PROGRAM MAIN
VAR
	// Control Buttons
	ManualSwitch: BOOL;
	AutoSwitch: BOOL;
	AutoStartButton: BOOL;
	ForwardSwitch: BOOL;
	ReverseSwitch: BOOL;
	StopSwitch: BOOL;
	
	// Limit switches
	LimitSwitchRight: BOOL;
	LimitSwitchLeft: BOOL;
	
	// Operation modes
	ManualMode: BOOL;
	AutoMode: BOOL;
	AutoStart: BOOL;
	ManualForward: BOOL;
	ManualReverse: BOOL;
	ConfirmAutoForward: BOOL;
	AutoForward: BOOL;
	AutoReverse: BOOL;
	
	// Output coils
	MotorForward: BOOL;
	MotorReverse: BOOL;
	
	// Aux. blocks
	tonForward: TON;
END_VAR
VAR // added by the converter: edge detectors and wires of the graphical bodies
    _w1 : BOOL;
END_VAR

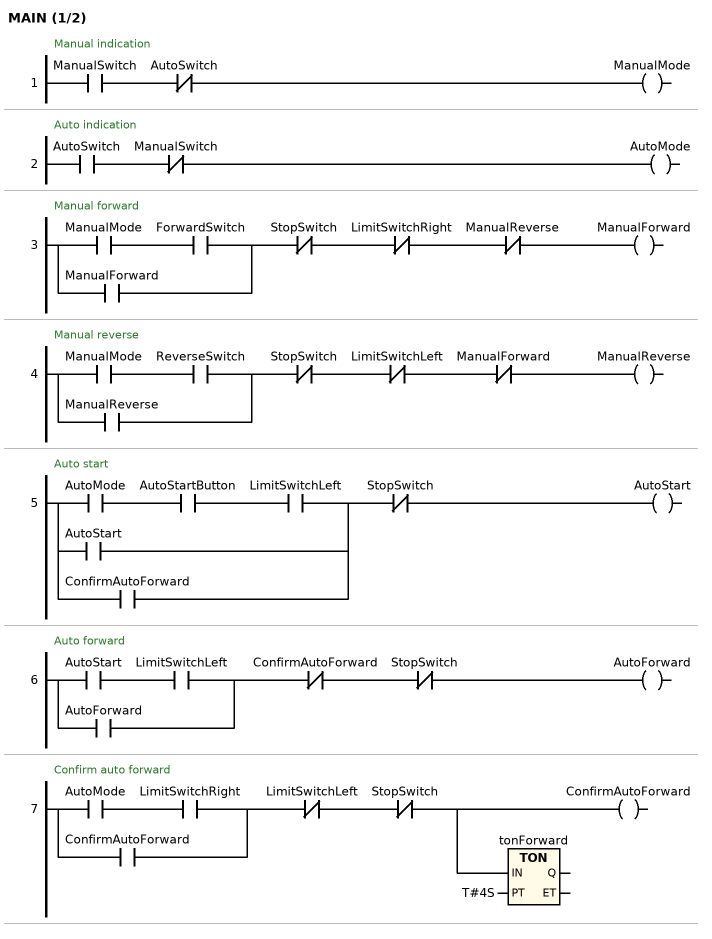
// NETWORK 1
// Manual indication
ManualMode := ManualSwitch AND NOT AutoSwitch;

// NETWORK 2
// Auto indication
AutoMode := AutoSwitch AND NOT ManualSwitch;

// NETWORK 3
// Manual forward
ManualForward := (ManualMode AND ForwardSwitch OR ManualForward) AND NOT StopSwitch AND NOT LimitSwitchRight AND NOT ManualReverse;

// NETWORK 4
// Manual reverse
ManualReverse := (ManualMode AND ReverseSwitch OR ManualReverse) AND NOT StopSwitch AND NOT LimitSwitchLeft AND NOT ManualForward;

// NETWORK 5
// Auto start
AutoStart := (AutoMode AND AutoStartButton AND LimitSwitchLeft OR AutoStart OR ConfirmAutoForward) AND NOT StopSwitch;

// NETWORK 6
// Auto forward
AutoForward := (AutoStart AND LimitSwitchLeft OR AutoForward) AND NOT ConfirmAutoForward AND NOT StopSwitch;

// NETWORK 7
// Confirm auto forward
_w1 := (AutoMode AND LimitSwitchRight OR ConfirmAutoForward) AND NOT LimitSwitchLeft AND NOT StopSwitch;
ConfirmAutoForward := _w1;
tonForward(IN := _w1, PT := T#4S); // TON

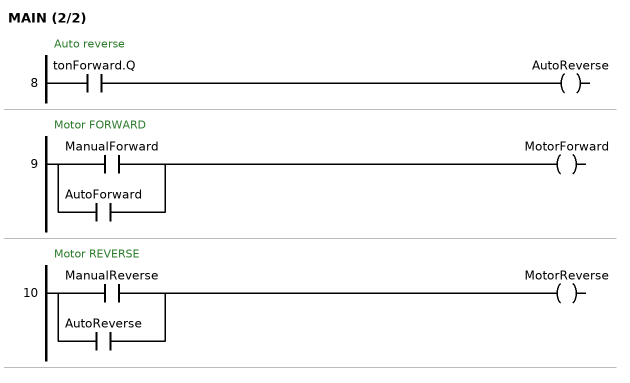
// NETWORK 8
// Auto reverse
AutoReverse := tonForward.Q;

// NETWORK 9
// Motor FORWARD
MotorForward := ManualForward OR AutoForward;

// NETWORK 10
// Motor REVERSE
MotorReverse := ManualReverse OR AutoReverse;

END_PROGRAM

(* stored: Version 1.1.0.1, ProductVersion 3.1.4024.15
   POU MAIN: Id {43a014b0-6970-4a8c-8fed-511ab9c87b1f}, SpecialFunc None *)
